FUNCTION_BLOCK FourStateDevice IMPLEMENTS I_FourStateDevice
VAR
	Q	AT%Q* : INT;
	_Status_prev	: INT;
END_VAR

METHOD Off

	Q	:=	REAL_TO_INT(F_Scaling(Variable_In:= 0, Input_min:= 0, Input_max:= 100, Output_min:= 0, Output_max:= 32767));
END_METHOD

METHOD On

	Q	:=	REAL_TO_INT(F_Scaling(Variable_In:= MAX(25, _Status_prev), Input_min:= 0, Input_max:= 100, Output_min:= 0, Output_max:= 32767));
END_METHOD

METHOD State_1

	Q	:=	REAL_TO_INT(F_Scaling(Variable_In:= 25, Input_min:= 0, Input_max:= 100, Output_min:= 0, Output_max:= 32767));
	_Status_prev	:=	25;
END_METHOD

METHOD State_2

	Q	:=	REAL_TO_INT(F_Scaling(Variable_In:= 50, Input_min:= 0, Input_max:= 100, Output_min:= 0, Output_max:= 32767));
	_Status_prev	:=	50;
END_METHOD

METHOD State_3

	Q	:=	REAL_TO_INT(F_Scaling(Variable_In:= 75, Input_min:= 0, Input_max:= 100, Output_min:= 0, Output_max:= 32767));
	_Status_prev	:=	75;
END_METHOD

METHOD State_4

	Q	:=	REAL_TO_INT(F_Scaling(Variable_In:= 100, Input_min:= 0, Input_max:= 100, Output_min:= 0, Output_max:= 32767));
	_Status_prev	:=	100;
END_METHOD

PROPERTY Status : INT
GET

	Status	:=	REAL_TO_INT(F_Scaling(Variable_In:= Q, Input_min:= 0, Input_max:= 32767, Output_min:= 0, Output_max:= 100));
END_GET
END_PROPERTY

END_FUNCTION_BLOCK

(* stored: Version 1.1.0.1, ProductVersion 3.1.4024.13
   POU FourStateDevice: Id {dea95f42-3b0e-4d09-a4bd-8a6267653bee}, SpecialFunc None
   Method Off: Id {b53edbde-d947-4e5f-b20f-0163f5cd9741}
   Method On: Id {aed5dade-2e33-450a-a330-304a67825435}
   Method State_1: Id {71392418-54dd-4aa0-bfc0-19a715638b51}
   Method State_2: Id {1faa0ff8-4586-4c03-acba-9e4b130277b7}
   Method State_3: Id {f00d21a5-063e-4727-b8d6-f9141ff82a71}
   Method State_4: Id {6118053d-9f8c-4874-8954-f8ac10f91b6d}
   Property Status: Id {5c938d1c-3a3a-48e0-9fe3-bab3ee0db1ba}
   Get Get: Id {17820d24-4d57-4131-9511-72385e032fd5} *)
